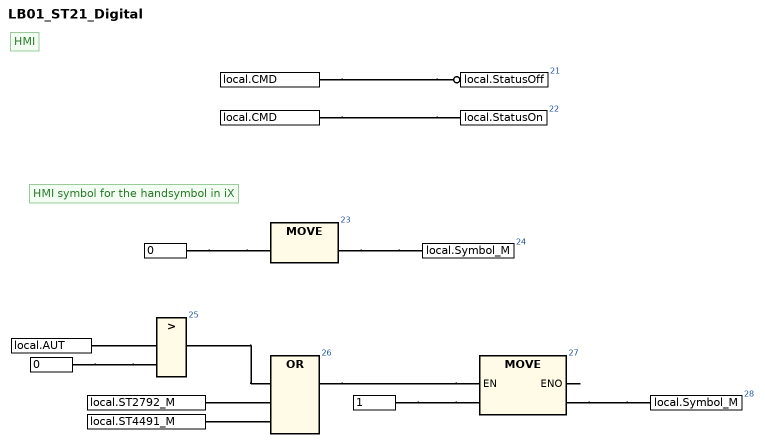
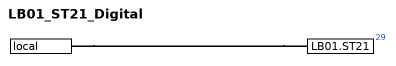
local := LB01.ST21;
sp1 := LB01.FF1.SP1;
operating := LB01.FF1.Operating;
nh_v := LB01.NH.V;
// Conditions for open.
delayST11(IN := LB01.GeneralStart, PT := DINT_TO_TIME(sp1 * 100)); // TON
local.CMD := (delayST11.Q OR operating AND NOT nh_v) AND local.AUT = 0 OR local.AUT = 2;
// Manual control from hardware switches
local.V := SEL(local.ST2792_M OR local.ST4491_M, local.CMD, SEL(local.ST2792_MCMD OR local.ST4491_OPM > 0.5 AND local.ST4491_M, FALSE, TRUE));
// HMI
local.StatusOff := NOT local.CMD;
local.StatusOn := local.CMD;
// HMI symbol for the handsymbol in iX
local.Symbol_M := 0;
IF local.AUT > 0 OR local.ST2792_M OR local.ST4491_M THEN _w1 := 1; END_IF
local.Symbol_M := _w1;
LB01.ST21 := local;

END_PROGRAM

// Device/AREA1/B001/LB01/Valve/SV61/LB01_SV61
PROGRAM LB01_SV61
VAR
	local:strValve;
	fbExercise: _BE_Exercise;
	FbAnalogOverride: _BE_AnalogueOverride;
	valueFreezeProtection: REAL;
	analogValue: REAL;
END_VAR
VAR // added by the converter: edge detectors and wires of the graphical bodies
    _w1, _w2 : BOOL;
    _w3, _w4, _w5 : ANY;
END_VAR

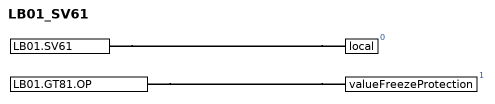
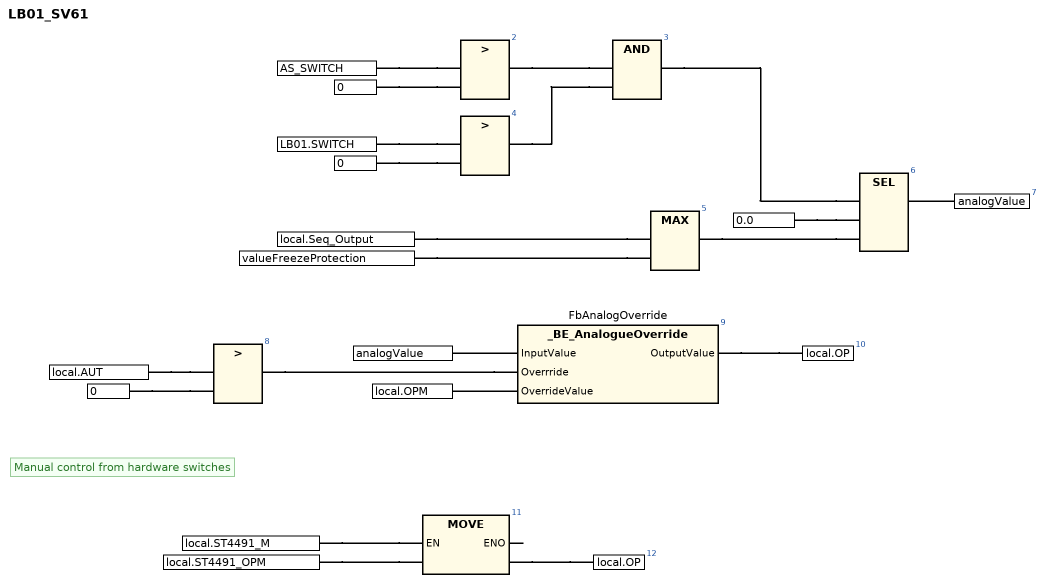
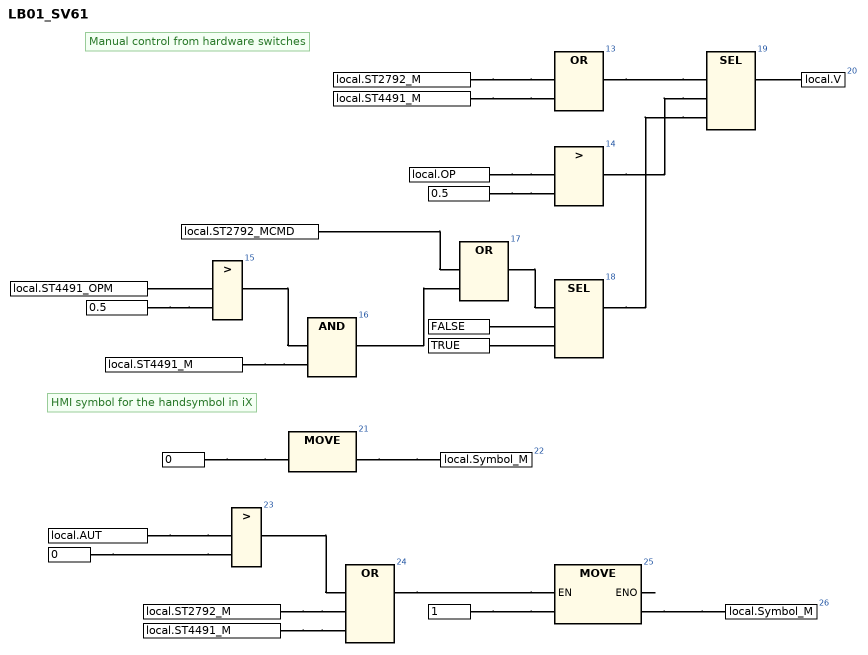
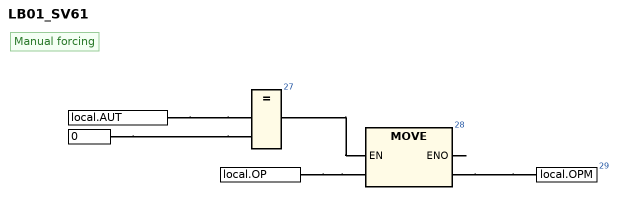
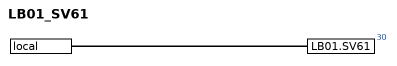
local := LB01.SV61;
valueFreezeProtection := LB01.GT81.OP;
_w2 := AS_SWITCH > 0 AND _w1;
_w1 := LB01.SWITCH > 0;
analogValue := SEL(_w2, 0.0, MAX(local.Seq_Output, valueFreezeProtection));
FbAnalogOverride(InputValue := analogValue, Overrride := local.AUT > 0, OverrideValue := local.OPM); // _BE_AnalogueOverride
local.OP := FbAnalogOverride.OutputValue;
// Manual control from hardware switches
IF local.ST4491_M THEN _w3 := local.ST4491_OPM; END_IF
local.OP := _w3;
// Manual control from hardware switches
local.V := SEL(local.ST2792_M OR local.ST4491_M, local.OP > 0.5, SEL(local.ST2792_MCMD OR local.ST4491_OPM > 0.5 AND local.ST4491_M, FALSE, TRUE));
// HMI symbol for the handsymbol in iX
local.Symbol_M := 0;
IF local.AUT > 0 OR local.ST2792_M OR local.ST4491_M THEN _w4 := 1; END_IF
local.Symbol_M := _w4;
// Manual forcing
IF local.AUT = 0 THEN _w5 := local.OP; END_IF
local.OPM := _w5;
LB01.SV61 := local;

END_PROGRAM

// Device/AREA1/B001/LB01/Valve/SV62/LB01_SV62
PROGRAM LB01_SV62
VAR
	local:strValve;
	FbAnalogueValve: _BE_AnalogueValve;
	fbExercise: _BE_Exercise;
	analogValue: REAL;
	valueFreezeProtection: REAL;
	FbAnalogOverride: _BE_AnalogueOverride;
END_VAR
VAR // added by the converter: edge detectors and wires of the graphical bodies
    _w1, _w2, _w3 : ANY;
END_VAR

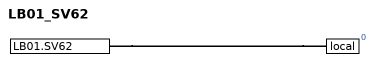
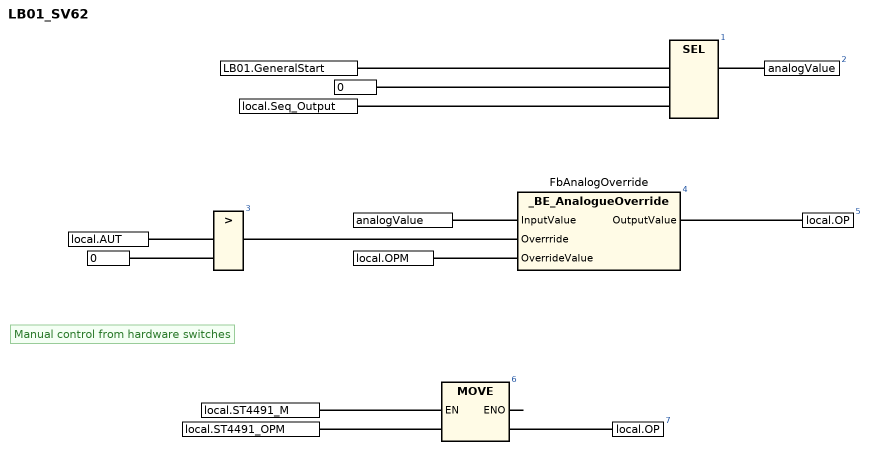
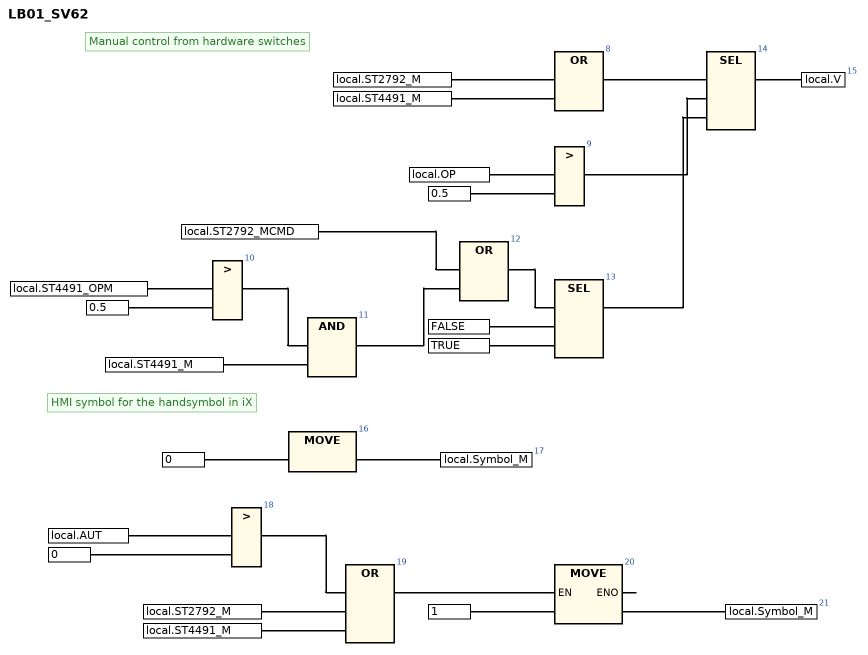
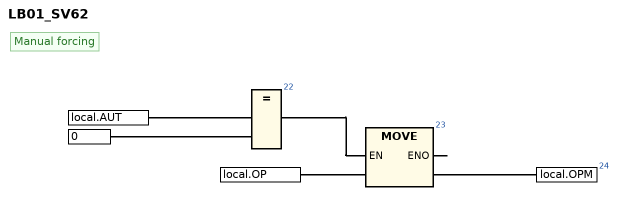
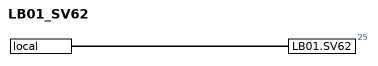
local := LB01.SV62;
analogValue := SEL(LB01.GeneralStart, 0, local.Seq_Output);
FbAnalogOverride(InputValue := analogValue, Overrride := local.AUT > 0, OverrideValue := local.OPM); // _BE_AnalogueOverride
local.OP := FbAnalogOverride.OutputValue;
// Manual control from hardware switches
IF local.ST4491_M THEN _w1 := local.ST4491_OPM; END_IF
local.OP := _w1;
// Manual control from hardware switches
local.V := SEL(local.ST2792_M OR local.ST4491_M, local.OP > 0.5, SEL(local.ST2792_MCMD OR local.ST4491_OPM > 0.5 AND local.ST4491_M, FALSE, TRUE));
// HMI symbol for the handsymbol in iX
local.Symbol_M := 0;
IF local.AUT > 0 OR local.ST2792_M OR local.ST4491_M THEN _w2 := 1; END_IF
local.Symbol_M := _w2;
// Manual forcing
IF local.AUT = 0 THEN _w3 := local.OP; END_IF
local.OPM := _w3;
LB01.SV62 := local;

END_PROGRAM

// Device/AREA1/B001/LB01/HeatExchanger/LB01_HeatExchanger_Rot
PROGRAM LB01_HeatExchanger_Rot
VAR
	local:strHeatExchanger_Rot;
	inputValue: LREAL;
	FbAnalogOverride: _BE_AnalogueOverride;
	inputAlarm: BOOL;
	nh_v: BOOL;
END_VAR
VAR // added by the converter: edge detectors and wires of the graphical bodies
    _w1, _w2, _w4, _w6, _w7 : ANY;
    _w3, _w5 : BOOL;
END_VAR

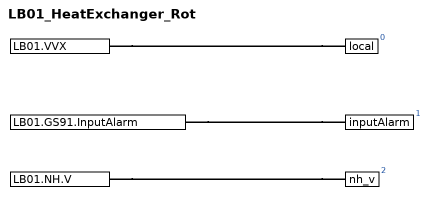
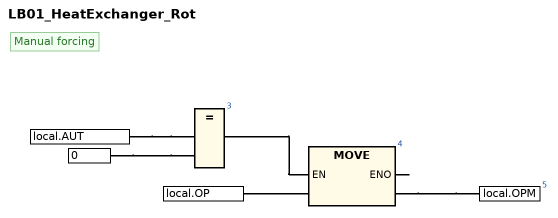
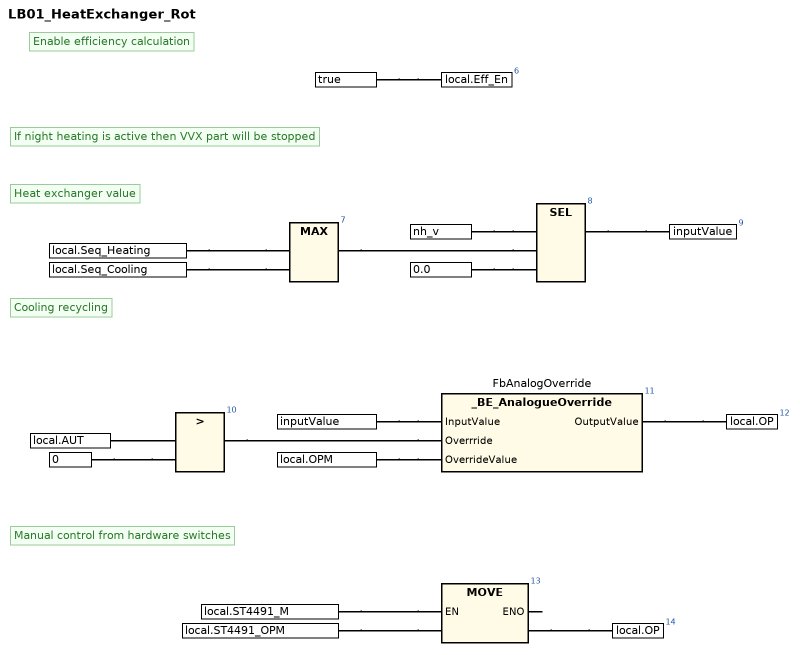
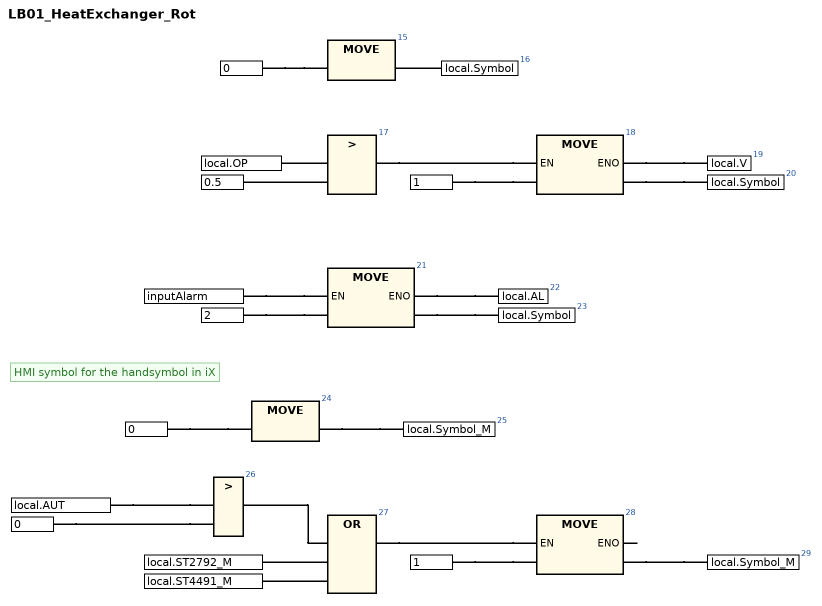
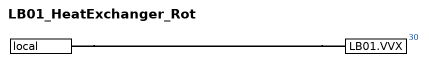
local := LB01.VVX;
inputAlarm := LB01.GS91.InputAlarm;
nh_v := LB01.NH.V;
// Manual forcing
IF local.AUT = 0 THEN _w1 := local.OP; END_IF
local.OPM := _w1;
// Enable efficiency calculation
local.Eff_En := true;
// If night heating is active then VVX part will be stopped
// Heat exchanger value
inputValue := SEL(nh_v, MAX(local.Seq_Heating, local.Seq_Cooling), 0.0);
// Cooling recycling
FbAnalogOverride(InputValue := inputValue, Overrride := local.AUT > 0, OverrideValue := local.OPM); // _BE_AnalogueOverride
local.OP := FbAnalogOverride.OutputValue;
// Manual control from hardware switches
IF local.ST4491_M THEN _w2 := local.ST4491_OPM; END_IF
local.OP := _w2;
local.Symbol := 0;
_w3 := local.OP > 0.5;
IF _w3 THEN _w4 := 1; END_IF
local.V := _w3;
local.Symbol := _w4;
_w5 := inputAlarm;
IF _w5 THEN _w6 := 2; END_IF
local.AL := _w5;
local.Symbol := _w6;
// HMI symbol for the handsymbol in iX
local.Symbol_M := 0;
IF local.AUT > 0 OR local.ST2792_M OR local.ST4491_M THEN _w7 := 1; END_IF
local.Symbol_M := _w7;
LB01.VVX := local;

END_PROGRAM

// Device/AREA1/B001/LB01/Sensor/Rotationguard/LB01_GS91
PROGRAM LB01_GS91
VAR
	local:strSensor6_HeatExchanger_Rot;
	AlarmAcknowledge01: _BE_AlarmAckRequired;
END_VAR
VAR // added by the converter: edge detectors and wires of the graphical bodies
    _w1, _w3 : ANY;
    _w2 : BOOL;
END_VAR

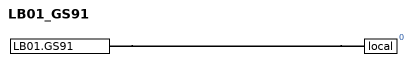
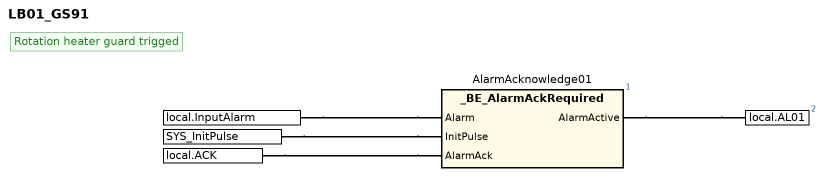
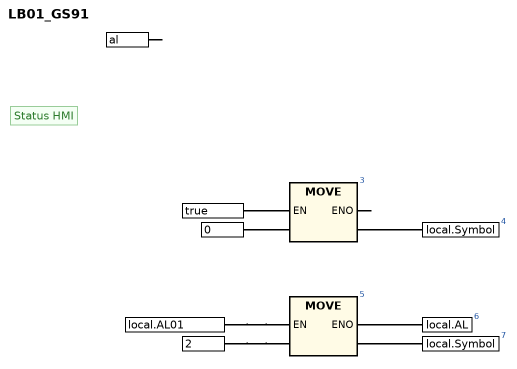
